// TIA Portal V19 export
FUNCTION "INPUT MAPPING" : Void   // FC3, LAD
{ S7_Optimized_Access := 'TRUE' }
// stored: SetENOAutomatically false
BEGIN

REGION Network 1: EMERGENCY STOP
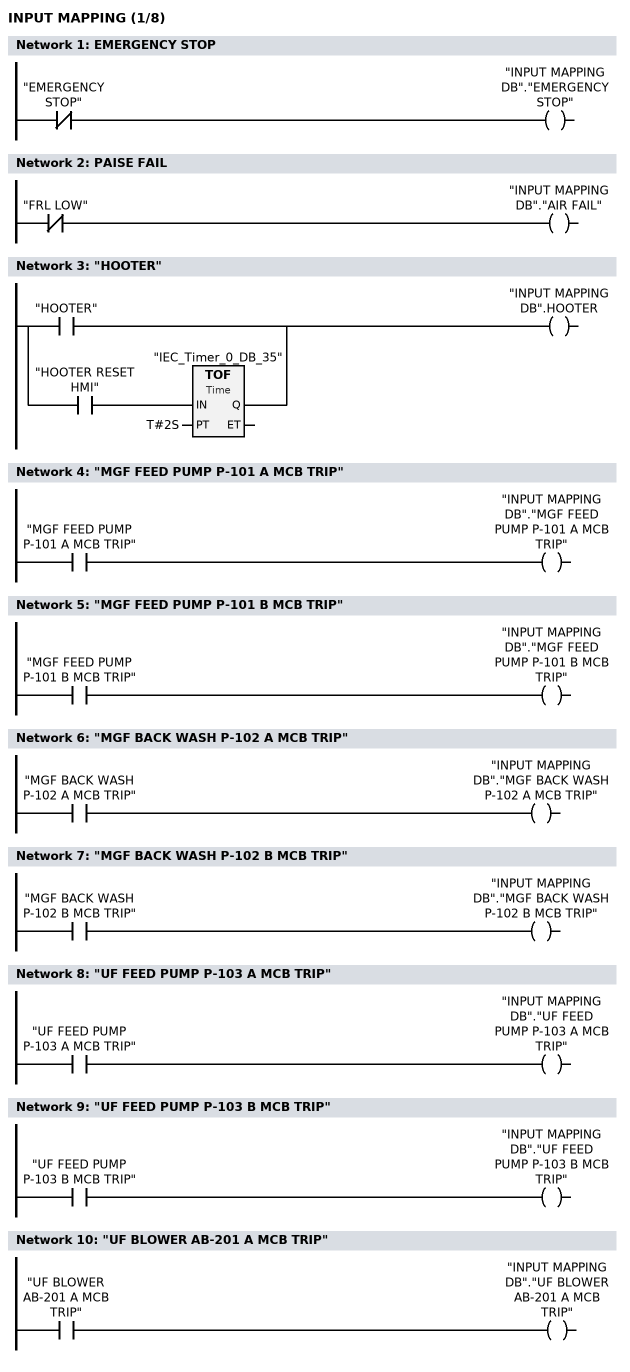
   RUNG wire#powerrail
      I_Contact( "EMERGENCY STOP" )
      Coil( "INPUT MAPPING DB"."EMERGENCY STOP" )
   END_RUNG
   // the same network as SCL:
   "INPUT MAPPING DB"."EMERGENCY STOP" := NOT "EMERGENCY STOP";
END_REGION

REGION Network 2: PAISE FAIL
   RUNG wire#powerrail
      I_Contact( "FRL LOW" )
      Coil( "INPUT MAPPING DB"."AIR FAIL" )
   END_RUNG
   // the same network as SCL:
   "INPUT MAPPING DB"."AIR FAIL" := NOT "FRL LOW";
END_REGION

REGION Network 3: "HOOTER"
   RUNG wire#powerrail
      Contact( "HOOTER" )
      wire#w1
      Coil( "INPUT MAPPING DB".HOOTER )
   END_RUNG
   RUNG wire#powerrail
      Contact( "HOOTER RESET HMI" )
      { S7_Templates := "time_type := Time" } "IEC_Timer_0_DB_35".TOF(pt := T#2S, et =>)
   END_RUNG wire#w1
   // the same network as SCL:
   "IEC_Timer_0_DB_35".TOF(IN := "HOOTER RESET HMI", PT := T#2S);
   "INPUT MAPPING DB".HOOTER := "HOOTER" OR "IEC_Timer_0_DB_35".Q;
END_REGION

REGION Network 4: "MGF FEED PUMP P-101 A MCB TRIP"
   RUNG wire#powerrail
      Contact( "MGF FEED PUMP P-101 A MCB TRIP" )
      Coil( "INPUT MAPPING DB"."MGF FEED PUMP P-101 A MCB TRIP" )
   END_RUNG
   // the same network as SCL:
   "INPUT MAPPING DB"."MGF FEED PUMP P-101 A MCB TRIP" := "MGF FEED PUMP P-101 A MCB TRIP";
END_REGION

REGION Network 5: "MGF FEED PUMP P-101 B MCB TRIP"
   RUNG wire#powerrail
      Contact( "MGF FEED PUMP P-101 B MCB TRIP" )
      Coil( "INPUT MAPPING DB"."MGF FEED PUMP P-101 B MCB TRIP" )
   END_RUNG
   // the same network as SCL:
   "INPUT MAPPING DB"."MGF FEED PUMP P-101 B MCB TRIP" := "MGF FEED PUMP P-101 B MCB TRIP";
END_REGION

REGION Network 6: "MGF BACK WASH P-102 A MCB TRIP"
   RUNG wire#powerrail
      Contact( "MGF BACK WASH  P-102 A MCB TRIP" )
      Coil( "INPUT MAPPING DB"."MGF BACK WASH  P-102 A MCB TRIP" )
   END_RUNG
   // the same network as SCL:
   "INPUT MAPPING DB"."MGF BACK WASH  P-102 A MCB TRIP" := "MGF BACK WASH  P-102 A MCB TRIP";
END_REGION

REGION Network 7: "MGF BACK WASH P-102 B MCB TRIP"
   RUNG wire#powerrail
      Contact( "MGF BACK WASH P-102 B MCB TRIP" )
      Coil( "INPUT MAPPING DB"."MGF BACK WASH P-102 B MCB TRIP" )
   END_RUNG
   // the same network as SCL:
   "INPUT MAPPING DB"."MGF BACK WASH P-102 B MCB TRIP" := "MGF BACK WASH P-102 B MCB TRIP";
END_REGION

REGION Network 8: "UF FEED PUMP P-103 A MCB TRIP"
   RUNG wire#powerrail
      Contact( "UF FEED PUMP P-103 A MCB TRIP" )
      Coil( "INPUT MAPPING DB"."UF FEED PUMP P-103 A MCB TRIP" )
   END_RUNG
   // the same network as SCL:
   "INPUT MAPPING DB"."UF FEED PUMP P-103 A MCB TRIP" := "UF FEED PUMP P-103 A MCB TRIP";
END_REGION

REGION Network 9: "UF FEED PUMP P-103 B MCB TRIP"
   RUNG wire#powerrail
      Contact( "UF FEED PUMP P-103 B MCB TRIP" )
      Coil( "INPUT MAPPING DB"."UF FEED PUMP P-103 B MCB TRIP" )
   END_RUNG
   // the same network as SCL:
   "INPUT MAPPING DB"."UF FEED PUMP P-103 B MCB TRIP" := "UF FEED PUMP P-103 B MCB TRIP";
END_REGION

REGION Network 10: "UF BLOWER AB-201 A MCB TRIP"
   RUNG wire#powerrail
      Contact( "UF BLOWER AB-201 A MCB TRIP" )
      Coil( "INPUT MAPPING DB"."UF BLOWER AB-201 A MCB TRIP" )
   END_RUNG
   // the same network as SCL:
   "INPUT MAPPING DB"."UF BLOWER AB-201 A MCB TRIP" := "UF BLOWER AB-201 A MCB TRIP";
END_REGION

REGION Network 11: "UF BLOWER AB-201 B MCB TRIP"
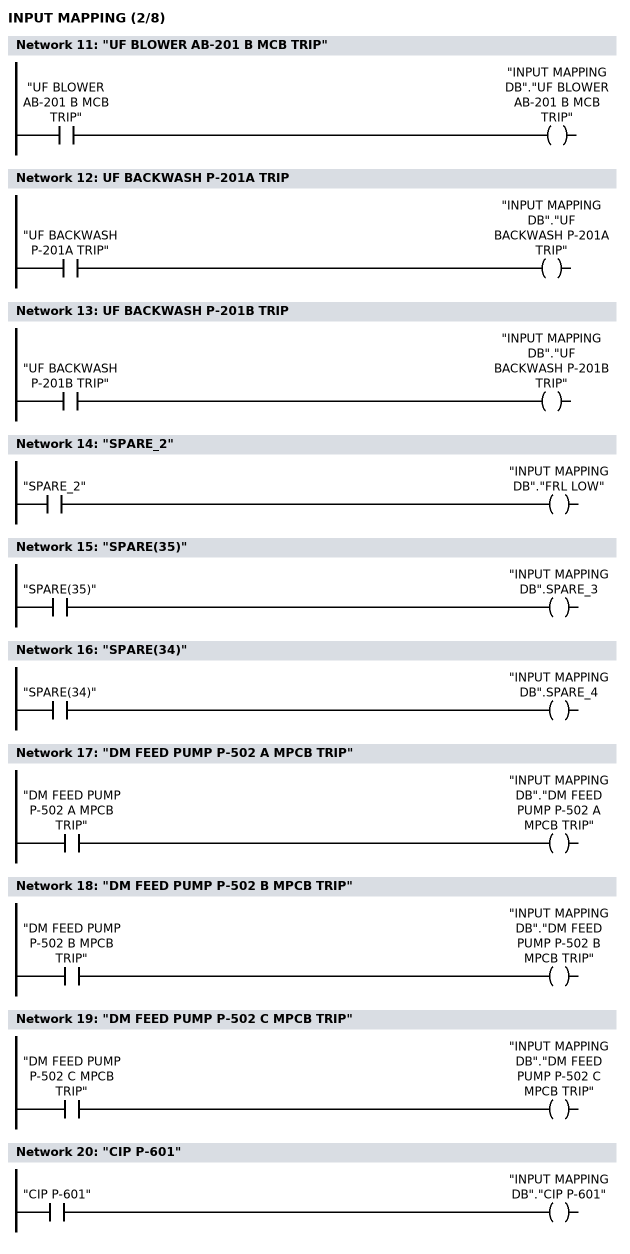
   RUNG wire#powerrail
      Contact( "UF BLOWER AB-201 B MCB TRIP" )
      Coil( "INPUT MAPPING DB"."UF BLOWER AB-201 B MCB TRIP" )
   END_RUNG
   // the same network as SCL:
   "INPUT MAPPING DB"."UF BLOWER AB-201 B MCB TRIP" := "UF BLOWER AB-201 B MCB TRIP";
END_REGION

REGION Network 12: UF BACKWASH P-201A TRIP
   RUNG wire#powerrail
      Contact( "UF BACKWASH P-201A TRIP" )
      Coil( "INPUT MAPPING DB"."UF BACKWASH P-201A TRIP" )
   END_RUNG
   // the same network as SCL:
   "INPUT MAPPING DB"."UF BACKWASH P-201A TRIP" := "UF BACKWASH P-201A TRIP";
END_REGION

REGION Network 13: UF BACKWASH P-201B TRIP
   RUNG wire#powerrail
      Contact( "UF BACKWASH P-201B TRIP" )
      Coil( "INPUT MAPPING DB"."UF BACKWASH P-201B TRIP" )
   END_RUNG
   // the same network as SCL:
   "INPUT MAPPING DB"."UF BACKWASH P-201B TRIP" := "UF BACKWASH P-201B TRIP";
END_REGION

REGION Network 14: "SPARE_2"
   RUNG wire#powerrail
      Contact( "SPARE_2" )
      Coil( "INPUT MAPPING DB"."FRL LOW" )
   END_RUNG
   // the same network as SCL:
   "INPUT MAPPING DB"."FRL LOW" := "SPARE_2";
END_REGION

REGION Network 15: "SPARE(35)"
   RUNG wire#powerrail
      Contact( "SPARE(35)" )
      Coil( "INPUT MAPPING DB".SPARE_3 )
   END_RUNG
   // the same network as SCL:
   "INPUT MAPPING DB".SPARE_3 := "SPARE(35)";
END_REGION

REGION Network 16: "SPARE(34)"
   RUNG wire#powerrail
      Contact( "SPARE(34)" )
      Coil( "INPUT MAPPING DB".SPARE_4 )
   END_RUNG
   // the same network as SCL:
   "INPUT MAPPING DB".SPARE_4 := "SPARE(34)";
END_REGION

REGION Network 17: "DM FEED PUMP P-502 A MPCB TRIP"
   RUNG wire#powerrail
      Contact( "DM FEED PUMP P-502 A MPCB TRIP" )
      Coil( "INPUT MAPPING DB"."DM FEED PUMP P-502 A MPCB TRIP" )
   END_RUNG
   // the same network as SCL:
   "INPUT MAPPING DB"."DM FEED PUMP P-502 A MPCB TRIP" := "DM FEED PUMP P-502 A MPCB TRIP";
END_REGION

REGION Network 18: "DM FEED PUMP P-502 B MPCB TRIP"
   RUNG wire#powerrail
      Contact( "DM FEED PUMP P-502 B MPCB TRIP" )
      Coil( "INPUT MAPPING DB"."DM FEED PUMP P-502 B MPCB TRIP" )
   END_RUNG
   // the same network as SCL:
   "INPUT MAPPING DB"."DM FEED PUMP P-502 B MPCB TRIP" := "DM FEED PUMP P-502 B MPCB TRIP";
END_REGION

REGION Network 19: "DM FEED PUMP P-502 C MPCB TRIP"
   RUNG wire#powerrail
      Contact( "DM FEED PUMP P-502 C MPCB TRIP" )
      Coil( "INPUT MAPPING DB"."DM FEED PUMP P-502 C MPCB TRIP" )
   END_RUNG
   // the same network as SCL:
   "INPUT MAPPING DB"."DM FEED PUMP P-502 C MPCB TRIP" := "DM FEED PUMP P-502 C MPCB TRIP";
END_REGION

REGION Network 20: "CIP P-601"
   RUNG wire#powerrail
      Contact( "CIP P-601" )
      Coil( "INPUT MAPPING DB"."CIP P-601" )
   END_RUNG
   // the same network as SCL:
   "INPUT MAPPING DB"."CIP P-601" := "CIP P-601";
END_REGION

REGION Network 21: "BACK WASH RECOVERY P-801 A MPCB TRIP"
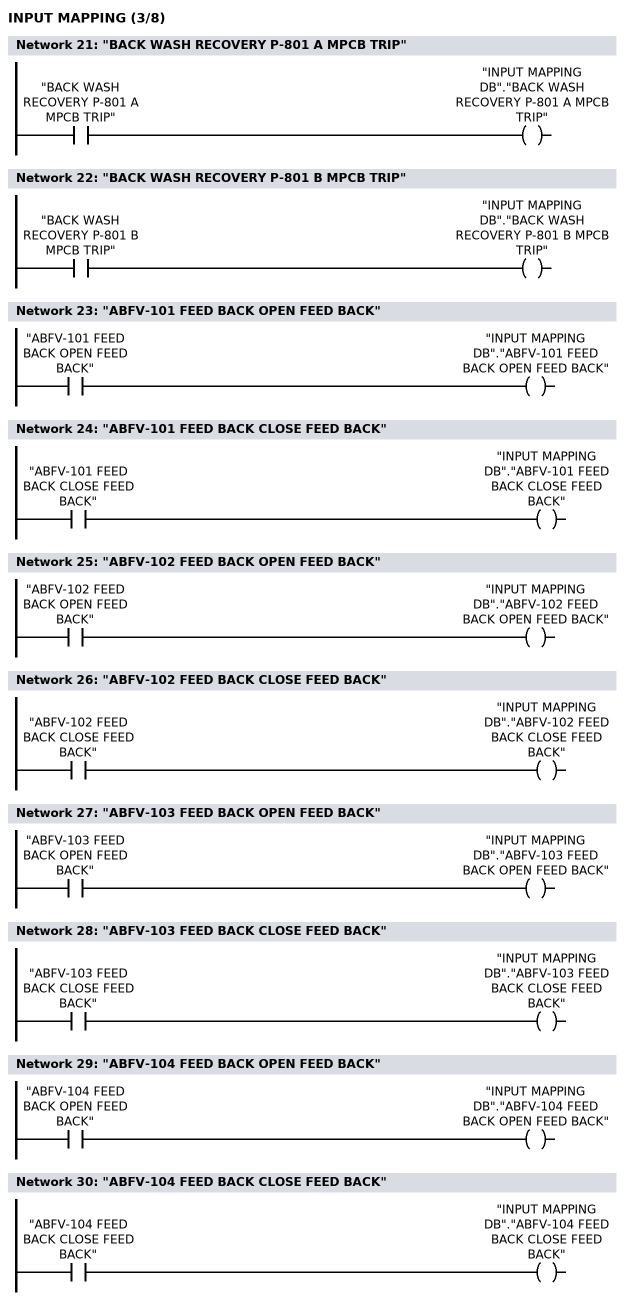
   RUNG wire#powerrail
      Contact( "BACK WASH RECOVERY P-801 A MPCB TRIP" )
      Coil( "INPUT MAPPING DB"."BACK WASH RECOVERY P-801 A MPCB TRIP" )
   END_RUNG
   // the same network as SCL:
   "INPUT MAPPING DB"."BACK WASH RECOVERY P-801 A MPCB TRIP" := "BACK WASH RECOVERY P-801 A MPCB TRIP";
END_REGION

REGION Network 22: "BACK WASH RECOVERY P-801 B MPCB TRIP"
   RUNG wire#powerrail
      Contact( "BACK WASH RECOVERY P-801 B MPCB TRIP" )
      Coil( "INPUT MAPPING DB"."BACK WASH RECOVERY P-801 B MPCB TRIP" )
   END_RUNG
   // the same network as SCL:
   "INPUT MAPPING DB"."BACK WASH RECOVERY P-801 B MPCB TRIP" := "BACK WASH RECOVERY P-801 B MPCB TRIP";
END_REGION

REGION Network 23: "ABFV-101 FEED BACK OPEN FEED BACK"
   RUNG wire#powerrail
      Contact( "ABFV-101 FEED BACK OPEN FEED BACK" )
      Coil( "INPUT MAPPING DB"."ABFV-101 FEED BACK OPEN FEED BACK" )
   END_RUNG
   // the same network as SCL:
   "INPUT MAPPING DB"."ABFV-101 FEED BACK OPEN FEED BACK" := "ABFV-101 FEED BACK OPEN FEED BACK";
END_REGION

REGION Network 24: "ABFV-101 FEED BACK CLOSE FEED BACK"
   RUNG wire#powerrail
      Contact( "ABFV-101 FEED BACK CLOSE FEED BACK" )
      Coil( "INPUT MAPPING DB"."ABFV-101 FEED BACK CLOSE FEED BACK" )
   END_RUNG
   // the same network as SCL:
   "INPUT MAPPING DB"."ABFV-101 FEED BACK CLOSE FEED BACK" := "ABFV-101 FEED BACK CLOSE FEED BACK";
END_REGION

REGION Network 25: "ABFV-102 FEED BACK OPEN FEED BACK"
   RUNG wire#powerrail
      Contact( "ABFV-102 FEED BACK OPEN FEED BACK" )
      Coil( "INPUT MAPPING DB"."ABFV-102 FEED BACK OPEN FEED BACK" )
   END_RUNG
   // the same network as SCL:
   "INPUT MAPPING DB"."ABFV-102 FEED BACK OPEN FEED BACK" := "ABFV-102 FEED BACK OPEN FEED BACK";
END_REGION

REGION Network 26: "ABFV-102 FEED BACK CLOSE FEED BACK"
   RUNG wire#powerrail
      Contact( "ABFV-102 FEED BACK CLOSE FEED BACK" )
      Coil( "INPUT MAPPING DB"."ABFV-102 FEED BACK CLOSE FEED BACK" )
   END_RUNG
   // the same network as SCL:
   "INPUT MAPPING DB"."ABFV-102 FEED BACK CLOSE FEED BACK" := "ABFV-102 FEED BACK CLOSE FEED BACK";
END_REGION

REGION Network 27: "ABFV-103 FEED BACK OPEN FEED BACK"
   RUNG wire#powerrail
      Contact( "ABFV-103 FEED BACK OPEN FEED BACK" )
      Coil( "INPUT MAPPING DB"."ABFV-103 FEED BACK OPEN FEED BACK" )
   END_RUNG
   // the same network as SCL:
   "INPUT MAPPING DB"."ABFV-103 FEED BACK OPEN FEED BACK" := "ABFV-103 FEED BACK OPEN FEED BACK";
END_REGION

REGION Network 28: "ABFV-103 FEED BACK CLOSE FEED BACK"
   RUNG wire#powerrail
      Contact( "ABFV-103 FEED BACK CLOSE FEED BACK" )
      Coil( "INPUT MAPPING DB"."ABFV-103 FEED BACK CLOSE FEED BACK" )
   END_RUNG
   // the same network as SCL:
   "INPUT MAPPING DB"."ABFV-103 FEED BACK CLOSE FEED BACK" := "ABFV-103 FEED BACK CLOSE FEED BACK";
END_REGION

REGION Network 29: "ABFV-104 FEED BACK OPEN FEED BACK"
   RUNG wire#powerrail
      Contact( "ABFV-104 FEED BACK OPEN FEED BACK" )
      Coil( "INPUT MAPPING DB"."ABFV-104 FEED BACK OPEN FEED BACK" )
   END_RUNG
   // the same network as SCL:
   "INPUT MAPPING DB"."ABFV-104 FEED BACK OPEN FEED BACK" := "ABFV-104 FEED BACK OPEN FEED BACK";
END_REGION

REGION Network 30: "ABFV-104 FEED BACK CLOSE FEED BACK"
   RUNG wire#powerrail
      Contact( "ABFV-104 FEED BACK CLOSE FEED BACK" )
      Coil( "INPUT MAPPING DB"."ABFV-104 FEED BACK CLOSE FEED BACK" )
   END_RUNG
   // the same network as SCL:
   "INPUT MAPPING DB"."ABFV-104 FEED BACK CLOSE FEED BACK" := "ABFV-104 FEED BACK CLOSE FEED BACK";
END_REGION

REGION Network 31: "ABFV 105 FEED BACK OPEN"
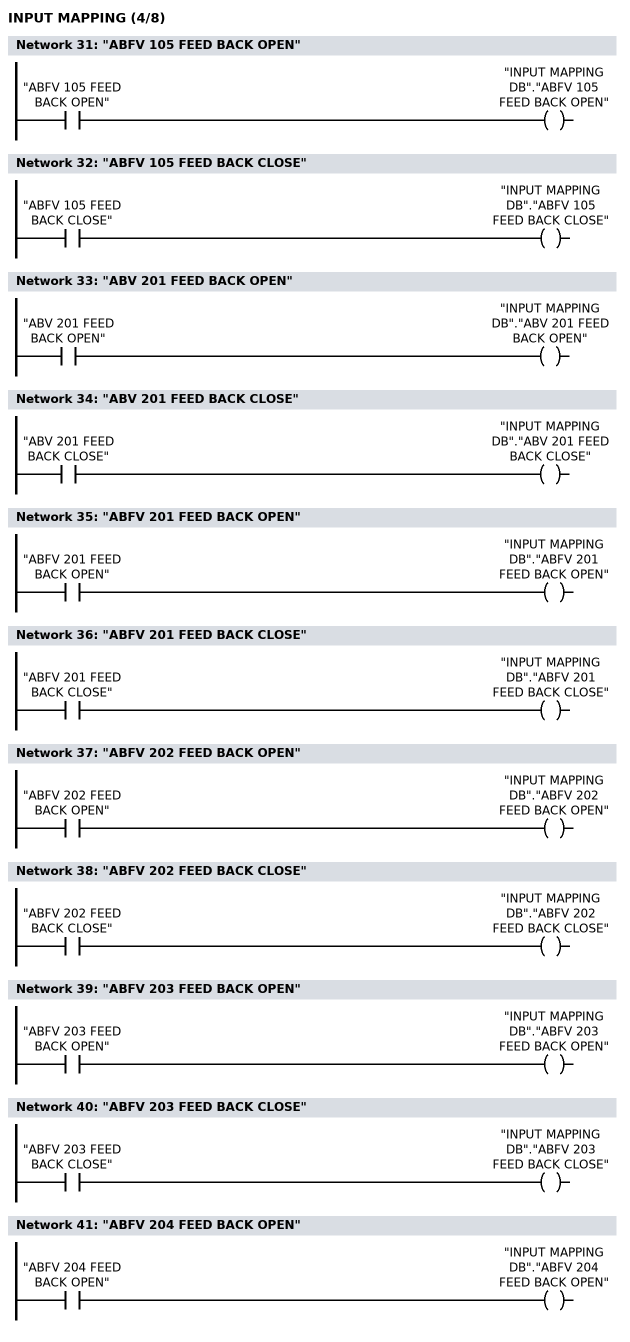
   RUNG wire#powerrail
      Contact( "ABFV 105 FEED BACK OPEN" )
      Coil( "INPUT MAPPING DB"."ABFV 105 FEED BACK OPEN" )
   END_RUNG
   // the same network as SCL:
   "INPUT MAPPING DB"."ABFV 105 FEED BACK OPEN" := "ABFV 105 FEED BACK OPEN";
END_REGION

REGION Network 32: "ABFV 105 FEED BACK CLOSE"
   RUNG wire#powerrail
      Contact( "ABFV 105 FEED BACK CLOSE" )
      Coil( "INPUT MAPPING DB"."ABFV 105 FEED BACK CLOSE" )
   END_RUNG
   // the same network as SCL:
   "INPUT MAPPING DB"."ABFV 105 FEED BACK CLOSE" := "ABFV 105 FEED BACK CLOSE";
END_REGION

REGION Network 33: "ABV 201 FEED BACK OPEN"
   RUNG wire#powerrail
      Contact( "ABV 201 FEED BACK OPEN" )
      Coil( "INPUT MAPPING DB"."ABV 201 FEED BACK OPEN" )
   END_RUNG
   // the same network as SCL:
   "INPUT MAPPING DB"."ABV 201 FEED BACK OPEN" := "ABV 201 FEED BACK OPEN";
END_REGION

REGION Network 34: "ABV 201 FEED BACK CLOSE"
   RUNG wire#powerrail
      Contact( "ABV 201 FEED BACK CLOSE" )
      Coil( "INPUT MAPPING DB"."ABV 201 FEED BACK CLOSE" )
   END_RUNG
   // the same network as SCL:
   "INPUT MAPPING DB"."ABV 201 FEED BACK CLOSE" := "ABV 201 FEED BACK CLOSE";
END_REGION

REGION Network 35: "ABFV 201 FEED BACK OPEN"
   RUNG wire#powerrail
      Contact( "ABFV 201 FEED BACK OPEN" )
      Coil( "INPUT MAPPING DB"."ABFV 201 FEED BACK OPEN" )
   END_RUNG
   // the same network as SCL:
   "INPUT MAPPING DB"."ABFV 201 FEED BACK OPEN" := "ABFV 201 FEED BACK OPEN";
END_REGION

REGION Network 36: "ABFV 201 FEED BACK CLOSE"
   RUNG wire#powerrail
      Contact( "ABFV 201 FEED BACK CLOSE" )
      Coil( "INPUT MAPPING DB"."ABFV 201 FEED BACK CLOSE" )
   END_RUNG
   // the same network as SCL:
   "INPUT MAPPING DB"."ABFV 201 FEED BACK CLOSE" := "ABFV 201 FEED BACK CLOSE";
END_REGION

REGION Network 37: "ABFV 202 FEED BACK OPEN"
   RUNG wire#powerrail
      Contact( "ABFV 202 FEED BACK OPEN" )
      Coil( "INPUT MAPPING DB"."ABFV 202 FEED BACK OPEN" )
   END_RUNG
   // the same network as SCL:
   "INPUT MAPPING DB"."ABFV 202 FEED BACK OPEN" := "ABFV 202 FEED BACK OPEN";
END_REGION

REGION Network 38: "ABFV 202 FEED BACK CLOSE"
   RUNG wire#powerrail
      Contact( "ABFV 202 FEED BACK CLOSE" )
      Coil( "INPUT MAPPING DB"."ABFV 202 FEED BACK CLOSE" )
   END_RUNG
   // the same network as SCL:
   "INPUT MAPPING DB"."ABFV 202 FEED BACK CLOSE" := "ABFV 202 FEED BACK CLOSE";
END_REGION

REGION Network 39: "ABFV 203 FEED BACK OPEN"
   RUNG wire#powerrail
      Contact( "ABFV 203 FEED BACK OPEN" )
      Coil( "INPUT MAPPING DB"."ABFV 203 FEED BACK OPEN" )
   END_RUNG
   // the same network as SCL:
   "INPUT MAPPING DB"."ABFV 203 FEED BACK OPEN" := "ABFV 203 FEED BACK OPEN";
END_REGION

REGION Network 40: "ABFV 203 FEED BACK CLOSE"
   RUNG wire#powerrail
      Contact( "ABFV 203 FEED BACK CLOSE" )
      Coil( "INPUT MAPPING DB"."ABFV 203 FEED BACK CLOSE" )
   END_RUNG
   // the same network as SCL:
   "INPUT MAPPING DB"."ABFV 203 FEED BACK CLOSE" := "ABFV 203 FEED BACK CLOSE";
END_REGION

REGION Network 41: "ABFV 204 FEED BACK OPEN"
   RUNG wire#powerrail
      Contact( "ABFV 204 FEED BACK OPEN" )
      Coil( "INPUT MAPPING DB"."ABFV 204 FEED BACK OPEN" )
   END_RUNG
   // the same network as SCL:
   "INPUT MAPPING DB"."ABFV 204 FEED BACK OPEN" := "ABFV 204 FEED BACK OPEN";
END_REGION

REGION Network 42: "ABFV 204 FEED BACK CLOSE"
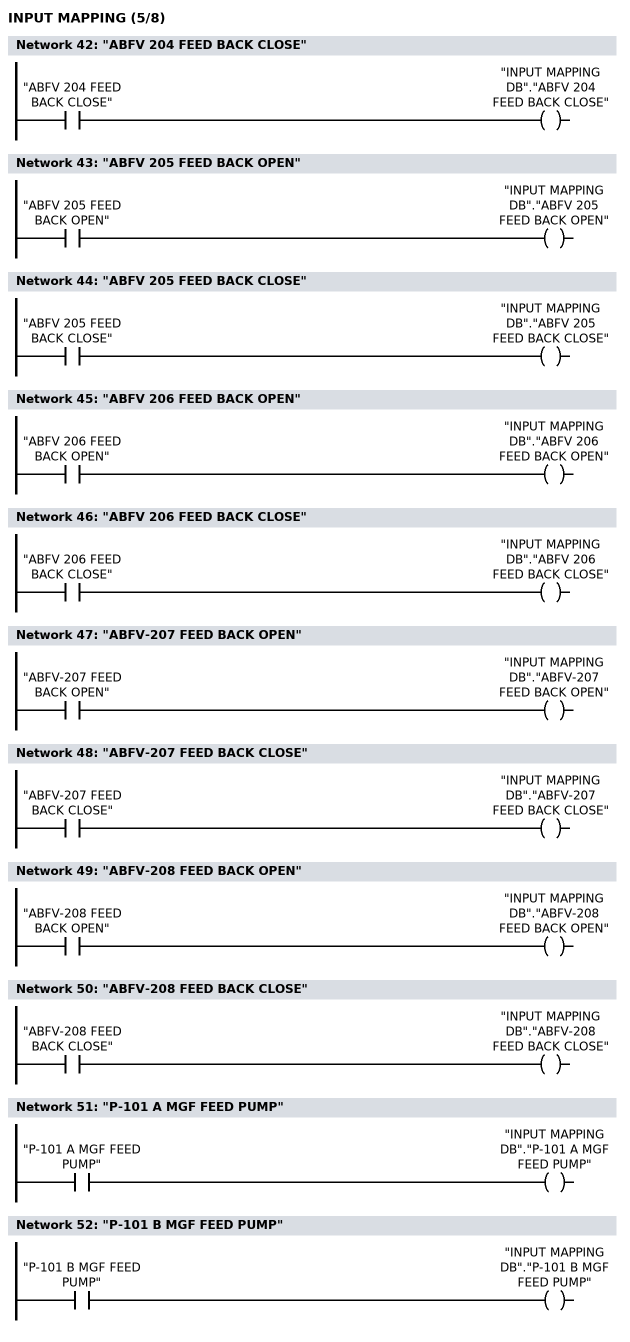
   RUNG wire#powerrail
      Contact( "ABFV 204 FEED BACK CLOSE" )
      Coil( "INPUT MAPPING DB"."ABFV 204 FEED BACK CLOSE" )
   END_RUNG
   // the same network as SCL:
   "INPUT MAPPING DB"."ABFV 204 FEED BACK CLOSE" := "ABFV 204 FEED BACK CLOSE";
END_REGION

REGION Network 43: "ABFV 205 FEED BACK OPEN"
   RUNG wire#powerrail
      Contact( "ABFV 205 FEED BACK OPEN" )
      Coil( "INPUT MAPPING DB"."ABFV 205 FEED BACK OPEN" )
   END_RUNG
   // the same network as SCL:
   "INPUT MAPPING DB"."ABFV 205 FEED BACK OPEN" := "ABFV 205 FEED BACK OPEN";
END_REGION

REGION Network 44: "ABFV 205 FEED BACK CLOSE"
   RUNG wire#powerrail
      Contact( "ABFV 205 FEED BACK CLOSE" )
      Coil( "INPUT MAPPING DB"."ABFV 205 FEED BACK CLOSE" )
   END_RUNG
   // the same network as SCL:
   "INPUT MAPPING DB"."ABFV 205 FEED BACK CLOSE" := "ABFV 205 FEED BACK CLOSE";
END_REGION

REGION Network 45: "ABFV 206 FEED BACK OPEN"
   RUNG wire#powerrail
      Contact( "ABFV 206 FEED BACK OPEN" )
      Coil( "INPUT MAPPING DB"."ABFV 206 FEED BACK OPEN" )
   END_RUNG
   // the same network as SCL:
   "INPUT MAPPING DB"."ABFV 206 FEED BACK OPEN" := "ABFV 206 FEED BACK OPEN";
END_REGION

REGION Network 46: "ABFV 206 FEED BACK CLOSE"
   RUNG wire#powerrail
      Contact( "ABFV 206 FEED BACK CLOSE" )
      Coil( "INPUT MAPPING DB"."ABFV 206 FEED BACK CLOSE" )
   END_RUNG
   // the same network as SCL:
   "INPUT MAPPING DB"."ABFV 206 FEED BACK CLOSE" := "ABFV 206 FEED BACK CLOSE";
END_REGION

REGION Network 47: "ABFV-207 FEED BACK OPEN"
   RUNG wire#powerrail
      Contact( "ABFV-207 FEED BACK OPEN" )
      Coil( "INPUT MAPPING DB"."ABFV-207 FEED BACK OPEN" )
   END_RUNG
   // the same network as SCL:
   "INPUT MAPPING DB"."ABFV-207 FEED BACK OPEN" := "ABFV-207 FEED BACK OPEN";
END_REGION

REGION Network 48: "ABFV-207 FEED BACK CLOSE"
   RUNG wire#powerrail
      Contact( "ABFV-207 FEED BACK CLOSE" )
      Coil( "INPUT MAPPING DB"."ABFV-207 FEED BACK CLOSE" )
   END_RUNG
   // the same network as SCL:
   "INPUT MAPPING DB"."ABFV-207 FEED BACK CLOSE" := "ABFV-207 FEED BACK CLOSE";
END_REGION

REGION Network 49: "ABFV-208 FEED BACK OPEN"
   RUNG wire#powerrail
      Contact( "ABFV-208 FEED BACK OPEN" )
      Coil( "INPUT MAPPING DB"."ABFV-208 FEED BACK OPEN" )
   END_RUNG
   // the same network as SCL:
   "INPUT MAPPING DB"."ABFV-208 FEED BACK OPEN" := "ABFV-208 FEED BACK OPEN";
END_REGION

REGION Network 50: "ABFV-208 FEED BACK CLOSE"
   RUNG wire#powerrail
      Contact( "ABFV-208 FEED BACK CLOSE" )
      Coil( "INPUT MAPPING DB"."ABFV-208 FEED BACK CLOSE" )
   END_RUNG
   // the same network as SCL:
   "INPUT MAPPING DB"."ABFV-208 FEED BACK CLOSE" := "ABFV-208 FEED BACK CLOSE";
END_REGION

REGION Network 51: "P-101 A MGF FEED PUMP"
   RUNG wire#powerrail
      Contact( "P-101 A MGF FEED PUMP" )
      Coil( "INPUT MAPPING DB"."P-101 A MGF FEED PUMP" )
   END_RUNG
   // the same network as SCL:
   "INPUT MAPPING DB"."P-101 A MGF FEED PUMP" := "P-101 A MGF FEED PUMP";
END_REGION

REGION Network 52: "P-101 B MGF FEED PUMP"
   RUNG wire#powerrail
      Contact( "P-101 B MGF FEED PUMP" )
      Coil( "INPUT MAPPING DB"."P-101 B MGF FEED PUMP" )
   END_RUNG
   // the same network as SCL:
   "INPUT MAPPING DB"."P-101 B MGF FEED PUMP" := "P-101 B MGF FEED PUMP";
END_REGION

REGION Network 53: "P-102 A MGF BACK WASH"
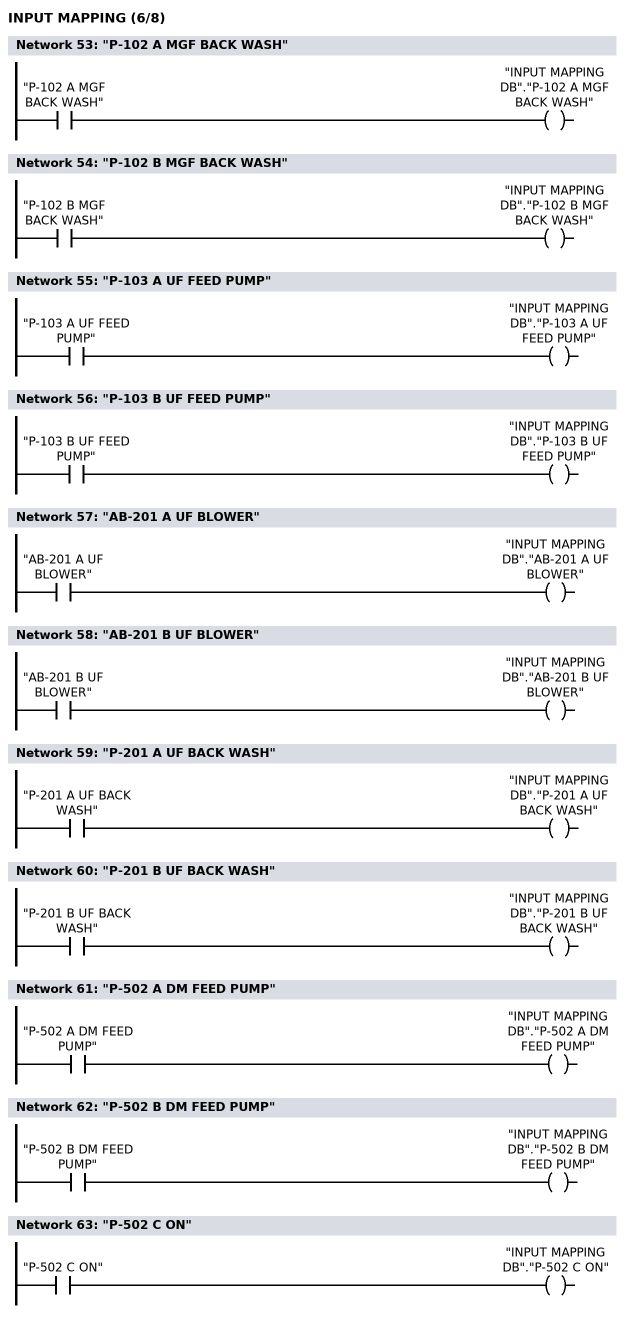
   RUNG wire#powerrail
      Contact( "P-102 A MGF BACK WASH" )
      Coil( "INPUT MAPPING DB"."P-102 A MGF BACK WASH" )
   END_RUNG
   // the same network as SCL:
   "INPUT MAPPING DB"."P-102 A MGF BACK WASH" := "P-102 A MGF BACK WASH";
END_REGION

REGION Network 54: "P-102 B MGF BACK WASH"
   RUNG wire#powerrail
      Contact( "P-102 B MGF BACK WASH" )
      Coil( "INPUT MAPPING DB"."P-102 B MGF BACK WASH" )
   END_RUNG
   // the same network as SCL:
   "INPUT MAPPING DB"."P-102 B MGF BACK WASH" := "P-102 B MGF BACK WASH";
END_REGION

REGION Network 55: "P-103 A UF FEED PUMP"
   RUNG wire#powerrail
      Contact( "P-103 A UF FEED PUMP" )
      Coil( "INPUT MAPPING DB"."P-103 A UF FEED PUMP" )
   END_RUNG
   // the same network as SCL:
   "INPUT MAPPING DB"."P-103 A UF FEED PUMP" := "P-103 A UF FEED PUMP";
END_REGION

REGION Network 56: "P-103 B UF FEED PUMP"
   RUNG wire#powerrail
      Contact( "P-103 B UF FEED PUMP" )
      Coil( "INPUT MAPPING DB"."P-103 B UF FEED PUMP" )
   END_RUNG
   // the same network as SCL:
   "INPUT MAPPING DB"."P-103 B UF FEED PUMP" := "P-103 B UF FEED PUMP";
END_REGION

REGION Network 57: "AB-201 A UF BLOWER"
   RUNG wire#powerrail
      Contact( "AB-201 A UF BLOWER" )
      Coil( "INPUT MAPPING DB"."AB-201 A UF BLOWER" )
   END_RUNG
   // the same network as SCL:
   "INPUT MAPPING DB"."AB-201 A UF BLOWER" := "AB-201 A UF BLOWER";
END_REGION

REGION Network 58: "AB-201 B UF BLOWER"
   RUNG wire#powerrail
      Contact( "AB-201 B UF BLOWER" )
      Coil( "INPUT MAPPING DB"."AB-201 B UF BLOWER" )
   END_RUNG
   // the same network as SCL:
   "INPUT MAPPING DB"."AB-201 B UF BLOWER" := "AB-201 B UF BLOWER";
END_REGION

REGION Network 59: "P-201 A UF BACK WASH"
   RUNG wire#powerrail
      Contact( "P-201 A UF BACK WASH" )
      Coil( "INPUT MAPPING DB"."P-201 A UF BACK WASH" )
   END_RUNG
   // the same network as SCL:
   "INPUT MAPPING DB"."P-201 A UF BACK WASH" := "P-201 A UF BACK WASH";
END_REGION

REGION Network 60: "P-201 B UF BACK WASH"
   RUNG wire#powerrail
      Contact( "P-201 B UF BACK WASH" )
      Coil( "INPUT MAPPING DB"."P-201 B UF BACK WASH" )
   END_RUNG
   // the same network as SCL:
   "INPUT MAPPING DB"."P-201 B UF BACK WASH" := "P-201 B UF BACK WASH";
END_REGION

REGION Network 61: "P-502 A DM FEED PUMP"
   RUNG wire#powerrail
      Contact( "P-502 A DM FEED PUMP" )
      Coil( "INPUT MAPPING DB"."P-502 A DM FEED PUMP" )
   END_RUNG
   // the same network as SCL:
   "INPUT MAPPING DB"."P-502 A DM FEED PUMP" := "P-502 A DM FEED PUMP";
END_REGION

REGION Network 62: "P-502 B DM FEED PUMP"
   RUNG wire#powerrail
      Contact( "P-502 B DM FEED PUMP" )
      Coil( "INPUT MAPPING DB"."P-502 B DM FEED PUMP" )
   END_RUNG
   // the same network as SCL:
   "INPUT MAPPING DB"."P-502 B DM FEED PUMP" := "P-502 B DM FEED PUMP";
END_REGION

REGION Network 63: "P-502 C ON"
   RUNG wire#powerrail
      Contact( "P-502 C ON" )
      Coil( "INPUT MAPPING DB"."P-502 C ON" )
   END_RUNG
   // the same network as SCL:
   "INPUT MAPPING DB"."P-502 C ON" := "P-502 C ON";
END_REGION

REGION Network 64: "P-601 ON"
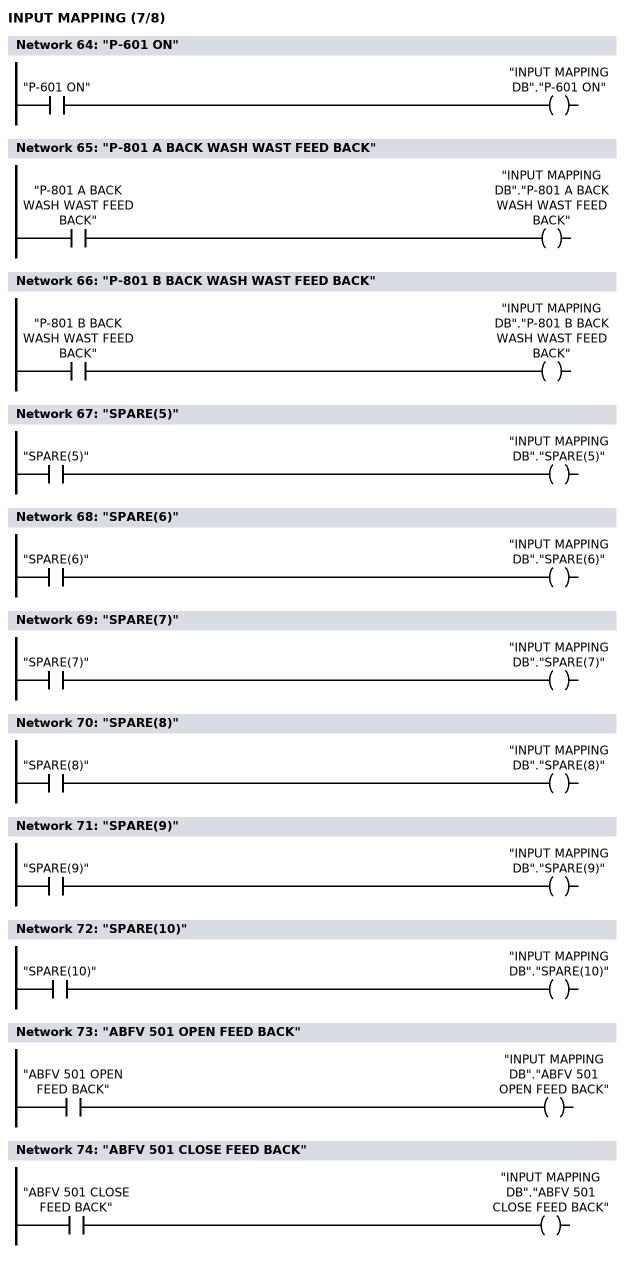
   RUNG wire#powerrail
      Contact( "P-601 ON" )
      Coil( "INPUT MAPPING DB"."P-601 ON" )
   END_RUNG
   // the same network as SCL:
   "INPUT MAPPING DB"."P-601 ON" := "P-601 ON";
END_REGION

REGION Network 65: "P-801 A BACK WASH WAST FEED BACK"
   RUNG wire#powerrail
      Contact( "P-801 A BACK WASH WAST FEED BACK" )
      Coil( "INPUT MAPPING DB"."P-801 A BACK WASH WAST FEED BACK" )
   END_RUNG
   // the same network as SCL:
   "INPUT MAPPING DB"."P-801 A BACK WASH WAST FEED BACK" := "P-801 A BACK WASH WAST FEED BACK";
END_REGION

REGION Network 66: "P-801 B BACK WASH WAST FEED BACK"
   RUNG wire#powerrail
      Contact( "P-801 B BACK WASH WAST FEED BACK" )
      Coil( "INPUT MAPPING DB"."P-801 B BACK WASH WAST FEED BACK" )
   END_RUNG
   // the same network as SCL:
   "INPUT MAPPING DB"."P-801 B BACK WASH WAST FEED BACK" := "P-801 B BACK WASH WAST FEED BACK";
END_REGION

REGION Network 67: "SPARE(5)"
   RUNG wire#powerrail
      Contact( "SPARE(5)" )
      Coil( "INPUT MAPPING DB"."SPARE(5)" )
   END_RUNG
   // the same network as SCL:
   "INPUT MAPPING DB"."SPARE(5)" := "SPARE(5)";
END_REGION

REGION Network 68: "SPARE(6)"
   RUNG wire#powerrail
      Contact( "SPARE(6)" )
      Coil( "INPUT MAPPING DB"."SPARE(6)" )
   END_RUNG
   // the same network as SCL:
   "INPUT MAPPING DB"."SPARE(6)" := "SPARE(6)";
END_REGION

REGION Network 69: "SPARE(7)"
   RUNG wire#powerrail
      Contact( "SPARE(7)" )
      Coil( "INPUT MAPPING DB"."SPARE(7)" )
   END_RUNG
   // the same network as SCL:
   "INPUT MAPPING DB"."SPARE(7)" := "SPARE(7)";
END_REGION

REGION Network 70: "SPARE(8)"
   RUNG wire#powerrail
      Contact( "SPARE(8)" )
      Coil( "INPUT MAPPING DB"."SPARE(8)" )
   END_RUNG
   // the same network as SCL:
   "INPUT MAPPING DB"."SPARE(8)" := "SPARE(8)";
END_REGION

REGION Network 71: "SPARE(9)"
   RUNG wire#powerrail
      Contact( "SPARE(9)" )
      Coil( "INPUT MAPPING DB"."SPARE(9)" )
   END_RUNG
   // the same network as SCL:
   "INPUT MAPPING DB"."SPARE(9)" := "SPARE(9)";
END_REGION

REGION Network 72: "SPARE(10)"
   RUNG wire#powerrail
      Contact( "SPARE(10)" )
      Coil( "INPUT MAPPING DB"."SPARE(10)" )
   END_RUNG
   // the same network as SCL:
   "INPUT MAPPING DB"."SPARE(10)" := "SPARE(10)";
END_REGION

REGION Network 73: "ABFV 501 OPEN FEED BACK"
   RUNG wire#powerrail
      Contact( "ABFV 501 OPEN FEED BACK" )
      Coil( "INPUT MAPPING DB"."ABFV 501 OPEN FEED BACK" )
   END_RUNG
   // the same network as SCL:
   "INPUT MAPPING DB"."ABFV 501 OPEN FEED BACK" := "ABFV 501 OPEN FEED BACK";
END_REGION

REGION Network 74: "ABFV 501 CLOSE FEED BACK"
   RUNG wire#powerrail
      Contact( "ABFV 501 CLOSE FEED BACK" )
      Coil( "INPUT MAPPING DB"."ABFV 501 CLOSE FEED BACK" )
   END_RUNG
   // the same network as SCL:
   "INPUT MAPPING DB"."ABFV 501 CLOSE FEED BACK" := "ABFV 501 CLOSE FEED BACK";
END_REGION

REGION Network 75: "ABFV 502 OPEN FEED BACK"
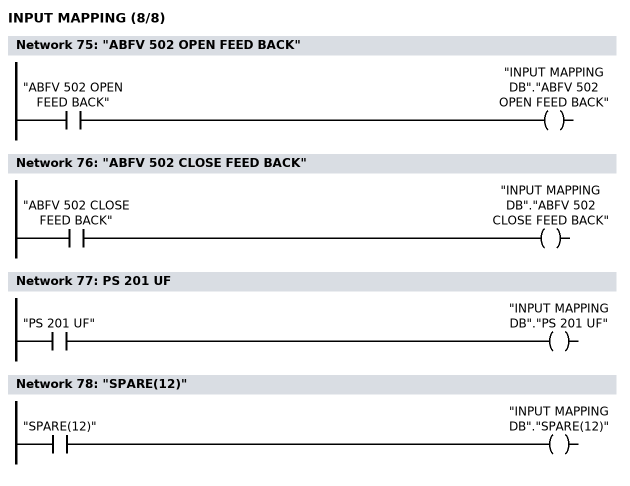
   RUNG wire#powerrail
      Contact( "ABFV 502 OPEN FEED BACK" )
      Coil( "INPUT MAPPING DB"."ABFV 502 OPEN FEED BACK" )
   END_RUNG
   // the same network as SCL:
   "INPUT MAPPING DB"."ABFV 502 OPEN FEED BACK" := "ABFV 502 OPEN FEED BACK";
END_REGION

REGION Network 76: "ABFV 502 CLOSE FEED BACK"
   RUNG wire#powerrail
      Contact( "ABFV 502 CLOSE FEED BACK" )
      Coil( "INPUT MAPPING DB"."ABFV 502 CLOSE FEED BACK" )
   END_RUNG
   // the same network as SCL:
   "INPUT MAPPING DB"."ABFV 502 CLOSE FEED BACK" := "ABFV 502 CLOSE FEED BACK";
END_REGION

REGION Network 77: PS 201 UF
   RUNG wire#powerrail
      Contact( "PS 201 UF" )
      Coil( "INPUT MAPPING DB"."PS 201 UF" )
   END_RUNG
   // the same network as SCL:
   "INPUT MAPPING DB"."PS 201 UF" := "PS 201 UF";
END_REGION

REGION Network 78: "SPARE(12)"
   RUNG wire#powerrail
      Contact( "SPARE(12)" )
      Coil( "INPUT MAPPING DB"."SPARE(12)" )
   END_RUNG
   // the same network as SCL:
   "INPUT MAPPING DB"."SPARE(12)" := "SPARE(12)";
END_REGION
END_FUNCTION
